Universal Robots PolyScope program: Tall_PHomeToInvD.urp

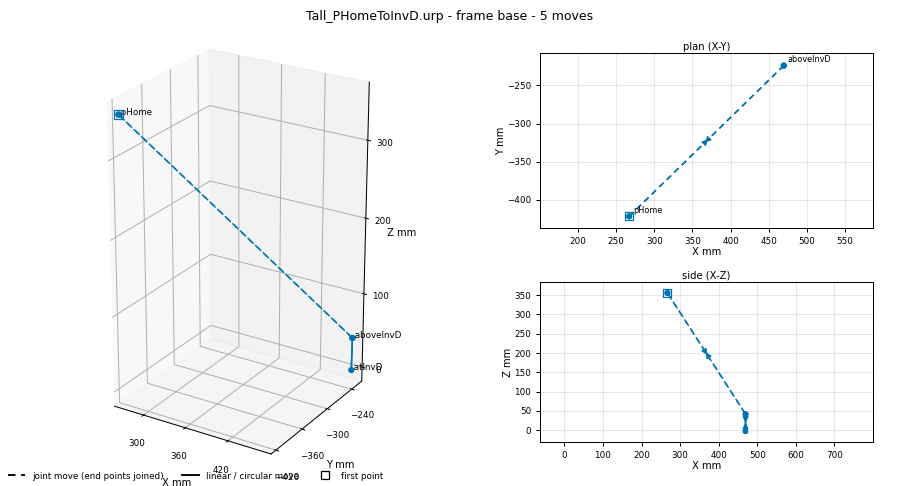
[picture p0: tool path of Tall_PHomeToInvD.urp in frame base, 5 of 5 moves have a stored position in this frame; points joined in program order, loops and branches not executed]
Program Tall_PHomeToInvD (installation=admin directory=/programs/THU_530PM/Final createdIn=3.8.0.61336 lastSavedIn=3.15.8.106339 robotSerialNumber=2015350924)
Calibrated DH parameters: a=[0, -0.425, -0.39225, 0, 0, 0]; d=[0.089159, 0, 0, 0.10915, 0.09465, 0.0823]; alpha=[1.570796, 0, 0, 1.570796, -1.570796, 0]; deltaTheta=[0, 0, 0, 0, 0, 0]
Robot Program (runOnlyOnce=true)
  Call _adminLinearIndex4
  MoveJ speed 180 deg/s, acceleration 200 deg/s^2 (useActiveTCP=true)
    Waypoint pHome: TCP in base x=267.143 y=-421.455 z=355.857 mm, rx=1.114 ry=1.106 rz=0.0051 rad; joints [-44.997, -90.001, -89.999, -90.001, 90.004, 0.008] deg; flange x=267.141 y=-421.459 z=431.857 mm, rx=-1.2021 ry=2.9025 rz=0.0001 rad
    Waypoint aboveInvD: motionParameters(blendRadius=0.043); TCP in base x=469.734 y=-223.868 z=41.581 mm, rx=1.706 ry=-0.0088 rz=-1.212 rad; joints [-13.348, -110.341, -116.782, -43.076, 89.918, 121.966] deg; flange x=470.016 y=-223.824 z=117.58 mm, rx=-1.2089 ry=-2.8962 rz=0.0031 rad
  MoveL speed 15 mm/s, acceleration 15 mm/s^2 (useActiveTCP=true) feature=Base
    Waypoint atInvD: TCP in base x=469.434 y=-224.17 z=-2.475 mm, rx=1.7059 ry=-0.0087 rz=-1.2121 rad; joints [-13.389, -115.496, -118.322, -36.388, 89.917, 121.924] deg; flange x=469.725 y=-224.127 z=73.524 mm, rx=-1.2089 ry=-2.8961 rz=0.0032 rad
    Set DigitalOutput pin=digital_out[0]; digitalValue=0
    Wait Sleep waitTime=1
    Waypoint aboveInvD: motionParameters(blendRadius=0.05); TCP in base x=469.734 y=-223.868 z=41.581 mm, rx=1.706 ry=-0.0088 rz=-1.212 rad; joints [-13.348, -110.341, -116.782, -43.076, 89.918, 121.966] deg; flange x=470.016 y=-223.824 z=117.58 mm, rx=-1.2089 ry=-2.8962 rz=0.0031 rad
  MoveJ speed 90 deg/s, acceleration 100 deg/s^2 (useActiveTCP=true)
    Waypoint pHome: TCP in base x=267.143 y=-421.455 z=355.857 mm, rx=1.114 ry=1.106 rz=0.0051 rad; joints [-44.997, -90.001, -89.999, -90.001, 90.004, 0.008] deg; flange x=267.141 y=-421.459 z=431.857 mm, rx=-1.2021 ry=2.9025 rz=0.0001 rad
SubProgram -> _adminLinearIndex4
SubProgram _adminLinearIndex4 (keepSynchronizedWithDisk=false) programFile=/programs/me345_admin/_adminLinearIndex4.urp
  Folder Move_linear_slide_Index4
    var_1 := False
    Loop While (checkContinuously=false) expression=var_1≟ False
      var_1 := socket_open("10.241.34.52",4001)
    var_3 := 1
    Send := "s r0x24 21"
    Script: socket_send_string(Send)
    Script: socket_send_byte(13)
    Send_Reply := socket_read_string()
    Send := "s r0xca 169167"
    Script: socket_send_string(Send)
    Script: socket_send_byte(13)
    Send_Reply := socket_read_string()
    Send := "t 1"
    Script: socket_send_string(Send)
    Script: socket_send_byte(13)
    Send_Reply := socket_read_string()
    Loop While (checkContinuously=false) expression=var_3≠0
      Send := "g r0xA0"
      Script: socket_send_string(Send)
      Script: socket_send_byte(13)
      var_3 := socket_get_var("v")
      Wait Sleep waitTime=0.1
    Script: socket_close()
    Script: sync()
